{attribute 'qualified_only'}
{attribute 'global_init_slot' := '50500'}
VAR_GLOBAL PERSISTENT
	//These tags are created here because you cannot write directly to local scoped tags(cpt_3144) from outside the POU
	//They are created here then mapped to the local variables in the POU
	//All tags in this GVL MUST have the {attribute 'OPC.UA.DA' :='1'} string above them in order to be exposed to OPC
	//Tags that are ONLY being read from the HMI have their values set in the opc_mapping program
		
	//State request INT from the HMI
	{attribute 'OPC.UA.DA' :='1'}
	popa_0200_hmi_state_request : INT;
	
	//Current Supervisor State
	{attribute 'OPC.UA.DA' :='1'}
	popa_0200_state : INT;
	
	//Current ED1 State
	{attribute 'OPC.UA.DA' :='1'}
	popa_0081_ed_state : INT;
	
	//ED1 Ok to transition from stop to idle
	{attribute 'OPC.UA.DA' :='1'}
	popa_0081_idle_transition_ok : BOOL;
	
	//ED1 Ok to transition from stop to CIP
	{attribute 'OPC.UA.DA' :='1'}
	popa_0081_cip_transition_ok : BOOL;
	
	//ED1 Ok to transition from stop to Manual
	{attribute 'OPC.UA.DA' :='1'}
	popa_0081_manual_transition_ok : BOOL;
	
	//ED1 Ok to transition from stop to Maintenance
	{attribute 'OPC.UA.DA' :='1'}
	popa_0081_maint_transition_ok : BOOL;
	
	//ED1 Ok to transition from idle to auto-input based
	{attribute 'OPC.UA.DA' :='1'}
	popa_0081_auto1_transition_ok : BOOL;
	
	//ED1 Ok to transition from idle to auto-concentration
	{attribute 'OPC.UA.DA' :='1'}
	popa_0081_auto2_transition_ok : BOOL;
	
	//ED1 Ok to transition from idle to auto-optimization
	{attribute 'OPC.UA.DA' :='1'}
	popa_0081_auto3_transition_ok : BOOL;
	
	//Pretreat Transfer State
	{attribute 'OPC.UA.DA' :='1'}
	popa_0070_state : INT;
	
	//Product Transfer State
	{attribute 'OPC.UA.DA' :='1'}
	popa_0120_state : INT;
	
	//Alarm Priority setpoint
	{attribute 'OPC.UA.DA' :='1'}
	popa_0081_cpt_3144_low_low_priority : INT;
	//Alarm delay setpoint(seconds)
	{attribute 'OPC.UA.DA' :='1'}
	popa_0081_cpt_3144_low_low_delay_setpoint : INT;
	//Alarm active for HMI
	{attribute 'OPC.UA.DA' :='1'}
	popa_0081_cpt_3144_low_low_active : BOOL;
	//Analog Alarm Setpoint
	{attribute 'OPC.UA.DA' :='1'}
	popa_0081_cpt_3144_low_low_setpoint : REAL;
	//Alarm enable
	{attribute 'OPC.UA.DA' :='1'}
	popa_0081_cpt_3144_low_low_enable: BOOL;
	
	//Alarm Priority setpoint
	{attribute 'OPC.UA.DA' :='1'}
	popa_0081_cpt_3144_low_priority : INT;
	//Alarm delay setpoint(seconds)
	{attribute 'OPC.UA.DA' :='1'}
	popa_0081_cpt_3144_low_delay_setpoint : INT;
	//Alarm active for HMI
	{attribute 'OPC.UA.DA' :='1'}
	popa_0081_cpt_3144_low_active : BOOL;
	//Analog Alarm Setpoint
	{attribute 'OPC.UA.DA' :='1'}
	popa_0081_cpt_3144_low_setpoint : REAL;
	//Alarm enable
	{attribute 'OPC.UA.DA' :='1'}
	popa_0081_cpt_3144_low_enable: BOOL;
	
	//Alarm Priority setpoint
	{attribute 'OPC.UA.DA' :='1'}
	popa_0081_cpt_3144_high_priority : INT;
	//Alarm delay setpoint(seconds)
	{attribute 'OPC.UA.DA' :='1'}
	popa_0081_cpt_3144_high_delay_setpoint : INT;
	//Alarm active for HMI
	{attribute 'OPC.UA.DA' :='1'}
	popa_0081_cpt_3144_high_active : BOOL;
	//Analog Alarm Setpoint
	{attribute 'OPC.UA.DA' :='1'}
	popa_0081_cpt_3144_high_setpoint : REAL;
	//Alarm enable
	{attribute 'OPC.UA.DA' :='1'}
	popa_0081_cpt_3144_high_enable: BOOL;
	
	//Alarm Priority setpoint
	{attribute 'OPC.UA.DA' :='1'}
	popa_0081_cpt_3144_high_high_priority : INT;
	//Alarm delay setpoint(seconds)
	{attribute 'OPC.UA.DA' :='1'}
	popa_0081_cpt_3144_high_high_delay_setpoint : INT;
	//Alarm active for HMI
	{attribute 'OPC.UA.DA' :='1'}
	popa_0081_cpt_3144_high_high_active : BOOL;
	//Analog Alarm Setpoint
	{attribute 'OPC.UA.DA' :='1'}
	popa_0081_cpt_3144_high_high_setpoint : REAL;
	//Alarm enable
	{attribute 'OPC.UA.DA' :='1'}
	popa_0081_cpt_3144_high_high_enable: BOOL;
	
	//System date time year
	{attribute 'OPC.UA.DA' :='1'}
	popa_0081_system_date_time_year : INT;
	//System date time month
	{attribute 'OPC.UA.DA' :='1'}
	popa_0081_system_date_time_month : INT;
	//System date time day
	{attribute 'OPC.UA.DA' :='1'}
	popa_0081_system_date_time_day : INT;
	//System date time hour
	{attribute 'OPC.UA.DA' :='1'}
	popa_0081_system_date_time_hour : INT;
	//System date time minute
	{attribute 'OPC.UA.DA' :='1'}
	popa_0081_system_date_time_minute : INT;
	//System date time second
	{attribute 'OPC.UA.DA' :='1'}
	popa_0081_system_date_time_second : INT;
	//Hour setpoint for daily reset triggers
	{attribute 'OPC.UA.DA' :='1'}
	popa_0081_daily_reset_hour_setpoint : INT;
	//Minute setpoint for daily reset triggers
	{attribute 'OPC.UA.DA' :='1'}
	popa_0081_daily_reset_minute_setpoint : INT;
	//Alarm acknowledge, acks all alarms, clears lower priority level alarms
	{attribute 'OPC.UA.DA' :='1'}
	popa_0081_alarm_ack : BOOL;
	//Alarm reset, clears higher priority alarms
	{attribute 'OPC.UA.DA' :='1'}
	popa_0081_alarm_reset : BOOL;
	
	//Raw Min value for analog input
	{attribute 'OPC.UA.DA' :='1'}
	popa_0081_cpt_3144_raw_min : REAL :=0;
	//Raw max value for analog input
	{attribute 'OPC.UA.DA' :='1'}
	popa_0081_cpt_3144_raw_max : REAL :=32767;
	//EU Min value for analog input
	{attribute 'OPC.UA.DA' :='1'}
	popa_0081_cpt_3144_eu_min : REAL;
	//EU Max value for analog input
	{attribute 'OPC.UA.DA' :='1'}
	popa_0081_cpt_3144_eu_max : REAL;
	//Filter factor value for analog input
	{attribute 'OPC.UA.DA' :='1'}
	popa_0081_cpt_3144_filter_factor : REAL;
	//Scaled value for analog input
	{attribute 'OPC.UA.DA' :='1'}
	popa_0081_cpt_3144_scaled_value : REAL;


END_VAR

(* stored: Version 1.1.0.1, ProductVersion 3.1.4024.12
   GVL opc: Id {674fd3be-a48d-4a85-a2e2-bd0824412020} *)
